Fanuc KAREL source: kt00492.KL

-- PROVISIONAL review KL for V940-1; original PC SHA256 3d3bb11f2322b39c38ec426351636c5f732ccbe0eac3e0e27ae23ee4eb71c677
-- Incomplete behavior may be omitted. Consult companion uncertainty JSON. Do not deploy.
PROGRAM KT00492
%NOLOCKGROUP
-- UNRESOLVED_DECL P1 type=000101
-- UNRESOLVED_DECL P2 type=000199
-- UNRESOLVED_DECL OUT type=000199
BEGIN
  -- V9_ZERO_TABLE_METADATA_HINT layout=0001; no indexed target words; source/name/runtime held
  -- UNRESOLVED_PC offsets 5-39; opcodes 49,49,7E,60,7E,4A
  -- UNRESOLVED_PC offsets 44-48; opcodes 7F
END KT00492
